ABB RobotStudio station: gofa_station.rsstn

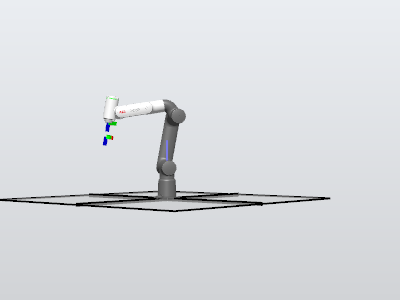
Station gofa_station (saved by RobotStudio 25.5.11605.0)
Controller Controller1
  mechanical unit ROB_1: CRB15000_5_95__02, 6 joints, base frame (0, 0, 0) mm
Layout (positions relative to the parent item):
  - CRB15000_5_95__02 [mechanism, from %ABB.RobotStudio.Models.CRB15000%\CRB15000_5_95__02.rslib] at (0, 0, 0) mm; joint values [2.5098, -0.1818, 0.353, 0.0037, 1.2324, -1.0491] (rad or m)
Targets, tools, work objects and paths stored in the station, written as RAPID:
! task T_ROB1
MODULE pick_and_place
  LOCAL PERS tooldata gripper:=[TRUE,[[0,0,117.85],[0.966,0,0,0.259]],[0.59,[0.15,0.01,57.98],[1,0,0,0],0,0,0]];
  LOCAL CONST robtarget HomePose:=[[-417.51,304.76,527.54],[0.04416,-0.99506,0.05359,0.07092],[1,-1,-1,0],[9E+09,9E+09,9E+09,9E+09,9E+09,9E+09]];
  LOCAL PROC GripClose()
    WaitTime 0.3;
  ENDPROC
  LOCAL PROC GripOpen()
    WaitTime 0.3;
  ENDPROC
  LOCAL PROC RunSession()
    MoveJ HomePose,v200,z50,gripper;
  ENDPROC
  PROC main()
    ConfJ \Off;
    ConfL \Off;
    MoveJ HomePose,v200,z50,gripper;
    GripOpen;
    RunSession;
  ENDPROC
ENDMODULE

! task T_ROB1
MODULE GOFA_ASI_Procedures
  PROC ASI_Routine2()
  ENDPROC
  PROC ASI_Routine1()
  ENDPROC
ENDMODULE

! task T_ROB1
MODULE Wizard_Params
  PROC wi_ProcPlaceHolder_Hidden()
  ENDPROC
ENDMODULE

